(* IEC 61131-3 sources: test/Class/_AccContCreateAdmin, 1 file *)

(* ---- _AccContCreateAdmin.st ---- *)
(*!
<Class
	Name               = "_AccContCreateAdmin"
	Revision           = "1.4"
	RealtimeTask       = "false"
	CyclicTask         = "false"
	BackgroundTask     = "false"
	Sigmatek           = "true"
	OSInterface        = "false"
	HighPriority       = "false"
	Automatic          = "false"
	UpdateMode         = "Prescan"
	SharedCommandTable = "true"
	Objectsize         = "(570,360)"
	Comment            = "class for creating a temporary admin">
	<Channels>
		<Server Name="ClassSvr" Visualized="false" Initialize="false" WriteProtected="true" Retentive="false" Comment="class server"/>
		<Server Name="Create" Visualized="false" Initialize="false" WriteProtected="false" Retentive="false" Comment="write() is the command for creating a Admin user"/>
		<Server Name="Level" Visualized="true" Initialize="true" WriteProtected="false" Retentive="false" Comment="user level default 255 (data channel)"/>
		<Server Name="PassWord" Visualized="true" Initialize="false" WriteProtected="false" Retentive="false" Comment="user password (channel to string object)"/>
		<Server Name="UserName" Visualized="true" Initialize="false" WriteProtected="false" Retentive="false" Comment="user name (channel to string object)"/>
		<Client Name="ccSystemLogging" Required="false" Internal="false" Comment="command channel to SystemLogging (optional)."/>
		<Client Name="coAccessControlMain" Required="true" Internal="false" Comment="object channel - Connect to AccessControlMain object"/>
		<Client Name="StrPassword" Required="true" Internal="true"/>
		<Client Name="StrUsername" Required="true" Internal="true"/>
	</Channels>
	<Dependencies>
		<Files>
			<File Path=".\Class\_AccContCreateAdmin\_AccContCreateAdmin_de.pdf"/>
			<File Path=".\Class\_AccContCreateAdmin\_AccContCreateAdmin_en.pdf"/>
		</Files>
	</Dependencies>
	<RevDoku>
		<Owner Company="Sigmatek"/>
		<Dokumentation Revision="1.4" Date="2016-10-10" Author="HubChr" Company="Sigmatek" Description="Added documentation pdfs."/>
		<Dokumentation Revision="1.3" Date="2016-10-05" Author="KaiAnd" Company="Sigmatek" Description="changed object channel for SystemLogging to a command channel; new help function LogMyText() for logging"/>
		<Dokumentation Revision="1.2" Date="2016-05-19" Author="GreJoh" Company="Sigmatek" Description="Client coSystemLogging need not be connected."/>
		<Dokumentation Revision="1.1" Date="2015-09-29" Author="BraLis" Company="Sigmatek" Description="insert the method SystemLogging::LogEventText instead of TRACE-Messages"/>
		<Dokumentation Revision="1.0" Date="2015-09-22" Company="Sigmatek" Description="Creation."/>
	</RevDoku>
	<Network Name="_AccContCreateAdmin">
		<!-- List of Components in this network -->
		<Components>
			<Object
				Name       = "StrPassword"
				Class      = "String"
				Position   = "(330,510)"
				Visualized = "true">
				<Channels>
					<Server Name="Data"/>
					<Client Name="SingleRealloc" Value="1"/>
				</Channels>
			</Object>
			<Object
				Name       = "StrUsername"
				Class      = "String"
				Position   = "(330,330)"
				Visualized = "true">
				<Channels>
					<Server Name="Data"/>
					<Client Name="SingleRealloc" Value="1"/>
				</Channels>
			</Object>
		</Components>
		<Comments>
		</Comments>
		<!-- List of Connections in this network -->
		<Connections>
			<Connection Source="this.StrUsername" Destination="StrUsername.Data"/>
			<Connection Source="this.StrPassword" Destination="StrPassword.Data"/>
			<Connection Source="this.UserName" Destination="StrUsername.Data" Vertices="(818,330),(646,420),"/>
			<Connection Source="this.PassWord" Destination="StrPassword.Data" Vertices="(818,390),(646,600),"/>
		</Connections>
		<!-- Headerfiles -->
		<Options>
		</Options>
	</Network>
</Class>
*)
_AccContCreateAdmin : CLASS
  //Servers:
	ClassSvr 	: SvrChCmd_DINT;
	Create 	: SvrCh_DINT;
	UserName 	: SvrCh_UDINT;
	PassWord 	: SvrCh_UDINT;
	Level 	: SvrCh_UDINT;
  //Clients:
	coAccessControlMain 	: CltChCmd__AccContMain;
	StrUsername 	: CltChCmd_String;
	StrPassword 	: CltChCmd_String;
	ccSystemLogging 	: CltChCmd_DINT;
  //Variables:
		IsCon_ccSystemLogging 	: BOOL;
  //Functions:

	FUNCTION VIRTUAL GLOBAL Init;
				//! <Function Comment="help function to log a text via command channel to SystemLogging" Name="LogMyText"/>
	FUNCTION LogMyText
		VAR_INPUT
			pLogTxt 	: ^CHAR;			//! <Variable Comment="pointer to the text which should be logged" Name="LogMyText.pLogTxt"/>
		END_VAR;

	FUNCTION VIRTUAL GLOBAL Create::Write
		VAR_INPUT
			input (EAX) 	: DINT;
		END_VAR
		VAR_OUTPUT
			result (EAX) 	: DINT;
		END_VAR;
  //Tables:
	FUNCTION @STD
		VAR_OUTPUT
			ret_code	: CONFSTATES;
		END_VAR;
	FUNCTION GLOBAL TAB @CT_;
END_CLASS;

#pragma using String
#pragma usingLtd _AccContMain

FUNCTION VIRTUAL GLOBAL _AccContCreateAdmin::Init

  if _FirstScan then

    //-----------------------------------------------------------------------------------------
    //  check client-connnections and set flags
    //-----------------------------------------------------------------------------------------
    if IsClientConnected(#ccSystemLogging) then
      IsCon_ccSystemLogging := TRUE;
    else
      IsCon_ccSystemLogging := FALSE;
    end_if;

  end_if;

END_FUNCTION

FUNCTION VIRTUAL GLOBAL _AccContCreateAdmin::Create::Write
	VAR_INPUT
		input (EAX) 	: DINT;
	END_VAR
	VAR_OUTPUT
		result (EAX) 	: DINT;
	END_VAR
  VAR
  	aTmpUsername : ARRAY[0..255] of CHAR;
    aTmpPassword : ARRAY[0..255] of CHAR;
    tmpLenUsername : UDINT;
    tmpLenPassword : UDINT;
  END_VAR

	Create := input;
	result := Create;

  tmpLenUsername := StrUsername.GetLength() + 1;
  tmpLenPassword:= StrPassword.GetLength() + 1;

  if tmpLenUsername > 0 then
    StrUsername.GetDataAt(pData:=#aTmpUsername[0], udSize:=tmpLenUsername, udAt:=0);
    StrPassword.GetDataAt(pData:=#aTmpPassword[0], udSize:=tmpLenPassword, udAt:=0);

    coAccessControlMain.CreateAdmin(pUsername:=#aTmpUsername[0], pPassword:=#aTmpPassword[0], usLevel:=to_usint(Level));
  else
    LogMyText("_AccContCreateAdmin::Create::Write: Kein User angelegt");

  end_if;

END_FUNCTION

FUNCTION _AccContCreateAdmin::LogMyText
VAR_INPUT
		pLogTxt 	: ^CHAR;
	END_VAR

  VAR
    NiGive	  : CmdStruct;
    NiGet     : Results;
  END_VAR

  if ((IsCon_ccSystemLogging = True) & (pLogTxt <> NIL)) then

    NiGive.uiCmd    := 0;               // Command
    NiGive.aPara[0] := (pLogTxt)$DINT;  // pointer to text

    ccSystemLogging.NewInst(#NiGive, #NiGet);

  end_if;

END_FUNCTION
